// TIA Portal V20 export
TYPE "LConSMC_typeKpAdaptionInput"
// stored: Access Published
   STRUCT
      enable : Bool;   // TRUE: Starte Funktionsbaustein / TRUE: Start function block
      adaptionMode : Bool;   // TRUE: Verwende Durchmesserverhältnis zur Adaption (dAct/dMax) FALSE: Verwende Trägheitsmomentverhältnis zur Adaption (JAct/JMax) / TRUE: User diameter ratio for adaption (dAct/dMax) FALSE: User inertia ratio for adaption (JAct/JMax)
      externalMode : Bool;   // TRUE: Adaptionswert wird nur berechnet aber nicht an den Antrieb gesendet (input "HWAddress" not needed) FALSE: Adaptionswert wird berechnet und an den Antrieb gesendet (Eingang "HWAddress" wird benötigt) / TRUE: Calculation of adaption value but value will not be written to telegram (input "HWAddress" not needed) FALSE: Adaption value will be calculated and written to the telegram (input "HWAddress" necessary)
      diameter : LReal;   // [m]/[inch] Aktueller Durchmesser / [m]/[inch] Current diameter
      HWAddress : HW_SUBMODULE;   // HW-Adresse des Telegramms über das der Adaptionswert an den Antrieb gesendet wird (nur wenn externalMode = FALSE) / HW-Address of telegram extension which is used to send adaption value to the drive (Only needed if externalMode = FALSE)
      offset : DInt := 6;   // Byte offset innerhalb des Telegramms für Kp-Adaptionswert (Wenn "externalMode" = FALSE). Wenn "offset" = 0 wird der Wert an den Anfang des Telegramms geschrieben / Byte offset with the telegram to write the Kp-Adaption value (if externalMode = FALSE). If "offset" = 0, the value will be written at the begining of the telegram
   END_STRUCT;
END_TYPE
